PROGRAM Log_Diverts_P2140
VAR
	r_DivertExtend			: ARRAY [1..16] OF R_TRIG;
	f_DivertExtend			: ARRAY [1..16] OF F_TRIG;
	r_ConfirmPE				: ARRAY [1..16] OF R_TRIG;
	f_ConfirmPE				: ARRAY [1..16] OF F_TRIG;
	sMessage				: STRING;
END_VAR

// Divert 1
r_DivertExtend[1](CLK := Sorter.aSorterDiverts_P2140[1].Output1);
f_DivertExtend[1](CLK := Sorter.aSorterDiverts_P2140[1].Output1);

IF r_DivertExtend[1].Q THEN
	IF .nDivertLogEnable.DIVERT1 THEN
		ADSLOGSTR( msgCtrlMask := ADSLOG_MSGTYPE_HINT OR ADSLOG_MSGTYPE_LOG
			, msgFmtStr := 'Extend Divert 1 : %s'
			, strArg := UDINT_TO_STRING(Sorter.st_SorterEncoder_P2140.CurrentCount)); 
	END_IF;
END_IF
IF f_DivertExtend[1].Q THEN
	IF .nDivertLogEnable.DIVERT1 THEN
		ADSLOGSTR( msgCtrlMask := ADSLOG_MSGTYPE_HINT OR ADSLOG_MSGTYPE_LOG
			, msgFmtStr := 'Retract Divert 1 : %s'
			, strArg := UDINT_TO_STRING(Sorter.st_SorterEncoder_P2140.CurrentCount)); 
	END_IF;
END_IF

// Confirm 1
r_ConfirmPE[1](CLK := Sorter.aSorterDiverts_P2140[1].ConfirmPE);
f_ConfirmPE[1](CLK := Sorter.aSorterDiverts_P2140[1].ConfirmPE);

IF r_ConfirmPE[1].Q THEN
	IF .nDivertLogEnable.CONFIRM1 THEN
		ADSLOGSTR( msgCtrlMask := ADSLOG_MSGTYPE_HINT OR ADSLOG_MSGTYPE_LOG
			, msgFmtStr := 'Confirm PE 1 Blocked: %s'
			, strArg := UDINT_TO_STRING(Sorter.st_SorterEncoder_P2140.CurrentCount)); 
	END_IF;
END_IF
IF f_ConfirmPE[1].Q THEN
	IF .nDivertLogEnable.CONFIRM1 THEN
		ADSLOGSTR( msgCtrlMask := ADSLOG_MSGTYPE_HINT OR ADSLOG_MSGTYPE_LOG
			, msgFmtStr := 'Confirm PE 1 Clear: %s'
			, strArg := UDINT_TO_STRING(Sorter.st_SorterEncoder_P2140.CurrentCount)); 
	END_IF;
END_IF

// Divert 2
r_DivertExtend[2](CLK := Sorter.aSorterDiverts_P2140[2].Output1);
f_DivertExtend[2](CLK := Sorter.aSorterDiverts_P2140[2].Output1);

IF r_DivertExtend[2].Q THEN
	IF .nDivertLogEnable.DIVERT2 THEN
		ADSLOGSTR( msgCtrlMask := ADSLOG_MSGTYPE_HINT OR ADSLOG_MSGTYPE_LOG
			, msgFmtStr := 'Extend Divert 2: %s'
			, strArg := UDINT_TO_STRING(Sorter.st_SorterEncoder_P2140.CurrentCount)); 
	END_IF;
END_IF
IF f_DivertExtend[2].Q THEN
	IF .nDivertLogEnable.DIVERT2 THEN
		ADSLOGSTR( msgCtrlMask := ADSLOG_MSGTYPE_HINT OR ADSLOG_MSGTYPE_LOG
			, msgFmtStr := 'Retract Divert 2: %s'
			, strArg := UDINT_TO_STRING(Sorter.st_SorterEncoder_P2140.CurrentCount)); 
	END_IF;
END_IF

// Confirm 2
r_ConfirmPE[2](CLK := Sorter.aSorterDiverts_P2140[2].ConfirmPE);
f_ConfirmPE[2](CLK := Sorter.aSorterDiverts_P2140[2].ConfirmPE);

IF r_ConfirmPE[2].Q THEN
	IF .nDivertLogEnable.CONFIRM2 THEN
		ADSLOGSTR( msgCtrlMask := ADSLOG_MSGTYPE_HINT OR ADSLOG_MSGTYPE_LOG
			, msgFmtStr := 'Confirm PE 2 Blocked: %s'
			, strArg := UDINT_TO_STRING(Sorter.st_SorterEncoder_P2140.CurrentCount)); 
	END_IF;
END_IF
IF f_ConfirmPE[2].Q THEN
	IF .nDivertLogEnable.CONFIRM2 THEN
		ADSLOGSTR( msgCtrlMask := ADSLOG_MSGTYPE_HINT OR ADSLOG_MSGTYPE_LOG
			, msgFmtStr := 'Confirm PE 2 Clear: %s'
			, strArg := UDINT_TO_STRING(Sorter.st_SorterEncoder_P2140.CurrentCount)); 
	END_IF
END_IF

END_PROGRAM

(* stored: Version 1.1.0.1, ProductVersion 3.1.4024.4
   POU Log_Diverts_P2140: Id {e9fe6440-b139-4cb5-add5-489bd6f224e0}, SpecialFunc None *)
